Staubli VAL3: _moveToScan.pgx

program _moveToScan()
begin
  // ============================================================================
  // CMD 2: 스캔 위치로 이동
  // ============================================================================
  cls()
  putln("* CMD "+ toString("", nCmdSignal) +": 스캔 위치로 이동")

  nStatusSignal = 0
  call _sendStatus()

  movej(jScan, tTool, mNomSpeed)
  waitEndMove()
  gotoxy(0,1)
  putln("* 스캔 위치 도달")

  call _sendJoint()

  nStatusSignal = 2
  call _sendStatus()

  gotoxy(0,8)
  putln("현재 상태값 : "+ toString("", nStatusSignal))
  putln("========================")
  putln("      명령 대기 중...")
  putln("========================")
end
